FUNCTION_BLOCK FieldsToPublishEvent (* Transform individual fields to an Arrowhead Publish Event *)
  (* Standard: 61499-2; Description: Copyright (c) 2019 fortiss GmbH This program and the accompanying materials are made available under the terms of the Eclipse Public License 2.0 which is available at https://www.eclipse.org/legal/epl-2.0/ SPDX-License-Identifier: EPL-2.0 *)
  (* Version 1.0, 2019-10-17, Cabral, fortiss GmbH *)
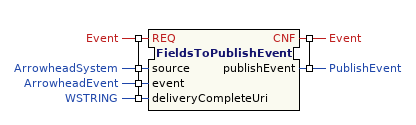
  EVENT_INPUT
    REQ WITH source, event, deliveryCompleteUri; (* Normal Execution Request *)
  END_EVENT
  EVENT_OUTPUT
    CNF WITH publishEvent; (* Execution Confirmation *)
  END_EVENT
  VAR_INPUT
    source : ArrowheadSystem; (* ArrowheadSystem publishing the event *)
    event : ArrowheadEvent; (* The published event *)
    deliveryCompleteUri : WSTRING; (* The URL subpath the Event Handler can use to inform the publisher about the results of the event propagation. If null, the Event Handler will not try to send the results *)
  END_VAR
  VAR_OUTPUT
    publishEvent : PublishEvent; (* Created publish event *)
  END_VAR
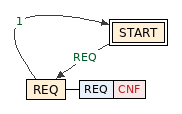
  EC_STATES
    START; (* Initial State *)
    REQ : REQ -> CNF;
  END_STATES
  EC_TRANSITIONS
    REQ TO START := 1;
    START TO REQ := REQ;
  END_TRANSITIONS
  ALGORITHM REQ IN ST: (* Initialization algorithm *)
publishEvent.source := source;
publishEvent.event := event;
publishEvent.deliveryCompleteUri := deliveryCompleteUri;
  END_ALGORITHM
END_FUNCTION_BLOCK
